// TIA Portal V16 export
// export: Created 2024-12-03T15:41:46.7047697Z, ExportSetting WithReadOnly, DisplayName Totally Integrated Automation Portal, DisplayVersion V16 Update 6, DisplayName TIA Portal Version Control Interface, DisplayVersion V16 Update 2, DisplayName TIA Portal Openness, DisplayVersion V16 Update 6, DisplayName TIA Portal Teamcenter Gateway, DisplayVersion V16, DisplayName SINAMICS Startdrive Advanced, DisplayVersion V16 Update 5, DisplayName SINAMICS Startdrive G130, G150, S120, S150, SINAMICS MV, S210, DisplayVersion V16 Update 5, DisplayName SINAMICS Startdrive G110M, G120, G120C, G120D, G120P, G115D, DisplayVersion V16 Update 5, DisplayName STEP 7 Professional, DisplayVersion V16 Update 6, DisplayName STEP 7 Safety, DisplayVersion V16, DisplayName WinCC Advanced / Unified PC, DisplayVersion V16 Update 6
VAR_GLOBAL   // PLC tag table "15 Scanners"
   I_Scan_100_ResultStatus AT %I1347.0 : "COGNEX_DATAMAN_IN_RESULT_STATUS_UDT";
   I_Scan_100_TriggerStatus AT %I1344.0 : "COGNEX_DATAMAN_IN_STATUS_UDT";
   I_Scan_100_ResultData AT %I1442.0 : "COGNEX_DATAMAN_IN_RESULT_UDT";
   Q_Scan_100_TriggerControl AT %Q1344.0 : "COGNEX_DATAMAN_OUT_TRIGGER_UDT";
   Q_Scan_100_ResultControl AT %Q1345.0 : "COGNEX_DATAMAN_OUT_CONTROL_UDT";
END_VAR
